// TIA Portal V19 export
DATA_BLOCK "LB212"   // DB149
// stored: InstanceOfName ButtonsSafe_LB212, InstanceOfType FB
"ButtonsSafe_LB212"
   // VAR_INPUT
   //    Reset_OthersPBs_Activation_IN : Bool;
   // END_VAR
   // VAR_OUTPUT
   //    Reset_OthersPBs_Activation_OUT : Bool;
   // END_VAR
   // VAR
   //    i : Int;
   //    iOperation : Int;
   //    iConcurrentOperation : Int;
   //    SettingWriteDone : Bool;
   //    PbPanel : "Buttons2Hands";
   //    PB : Struct
   //       ResetAlarms : Bool;
   //       DieClamp_Rest : Bool;
   //       DieClamp_Work : Bool;
   //       DieT1CutHead_Rest : Bool;
   //       DieT1CutHead_Work : Bool;
   //       DieT2MarkHead_Rest : Bool;
   //       DieT2MarkHead_Work : Bool;
   //       DieT3MarkHead_Rest : Bool;
   //       DieT3MarkHead_Work : Bool;
   //       Carriage_Bwd : Bool;
   //       Carriage_Fwd : Bool;
   //    END_STRUCT;
   // END_VAR
BEGIN
END_DATA_BLOCK
